(* IEC 61131-3 sources: test/Class/HmiBaseList, 1 file *)

(* ---- HmiBaseList.st ---- *)
(*!
<Class
	Name               = "HmiBaseList"
	Revision           = "0.0"
	RealtimeTask       = "false"
	CyclicTask         = "false"
	BackgroundTask     = "false"
	Sigmatek           = "true"
	OSInterface        = "false"
	HighPriority       = "false"
	Automatic          = "false"
	UpdateMode         = "Prescan"
	SharedCommandTable = "true"
	Objectsize         = "(284,120)">
	<Channels>
		<Server Name="ClassSvr" Visualized="false" Initialize="false" WriteProtected="true" Retentive="false"/>
		<Client Name="File" Required="true" Internal="false"/>
	</Channels>
</Class>
*)
HmiBaseList : CLASS
  //Servers:
	ClassSvr 	: SvrChCmd_DINT;
  //Clients:
	File 	: CltChCmd_HmiFile;
  //Variables:
  //Functions:

	FUNCTION GLOBAL LoadFile
		VAR_INPUT
			dpne 	: ^CHAR;
		END_VAR
		VAR_OUTPUT
			retcode 	: BOOL;
		END_VAR;

	FUNCTION VIRTUAL Load
		VAR_OUTPUT
			retcode 	: BOOL;
		END_VAR;

	FUNCTION VIRTUAL Free;
  //Tables:
	FUNCTION @STD
		VAR_OUTPUT
			ret_code	: CONFSTATES;
		END_VAR;
	FUNCTION GLOBAL TAB @CT_;
END_CLASS;

#pragma usingLtd HmiFile

FUNCTION VIRTUAL HmiBaseList::Free

END_FUNCTION

FUNCTION VIRTUAL HmiBaseList::Load
	VAR_OUTPUT
		retcode 	: BOOL;
	END_VAR

  retcode := false;

END_FUNCTION

FUNCTION GLOBAL HmiBaseList::LoadFile
	VAR_INPUT
		dpne 	: ^CHAR;
	END_VAR
	VAR_OUTPUT
		retcode 	: BOOL;
	END_VAR

  Free();
  retcode := false;

  if(File.FOpen(dpne, 'R') = true) then
    File.FReadHeader();
    retcode := Load(); // load imageinfo
    File.FClose();
  end_if;

END_FUNCTION
